ADAPTER ATimeOut (* Interface for a time out service roughly based on the definitions of ROOM *)
  (* Standard: 61499-1 *)
  (* Version 1.0, 2012-12-18, AZ, 4DIAC-Consortium *)
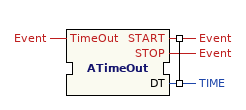
  EVENT_INPUT
    TimeOut; (* Request from Socket *)
  END_EVENT
  EVENT_OUTPUT
    START WITH DT; (* start timeout notifcation *)
    STOP; (* stop timeout notification *)
  END_EVENT
  VAR_OUTPUT
    DT : TIME; (* timeout duration *)
  END_VAR
  SERVICE SOCKET/PLUG (* Interface for a time out service roughly based on the definitions of ROOM *)
    SEQUENCE Timeout
      PLUG.START(TD) -> SOCKET.START(TD);
      SOCKET.TimeOut() -> PLUG.TimeOut();
    END_SEQUENCE
    SEQUENCE normal operation
      PLUG.Start(TD) -> SOCKET.Start(TD);
      PLUG.STOP() -> SOCKET.STOP();
    END_SEQUENCE
  END_SERVICE
END_ADAPTER
